// Mitsubishi GX Works2 project: miniproject_finalcode   PLC: Q03UDV

PROGRAM MAIN
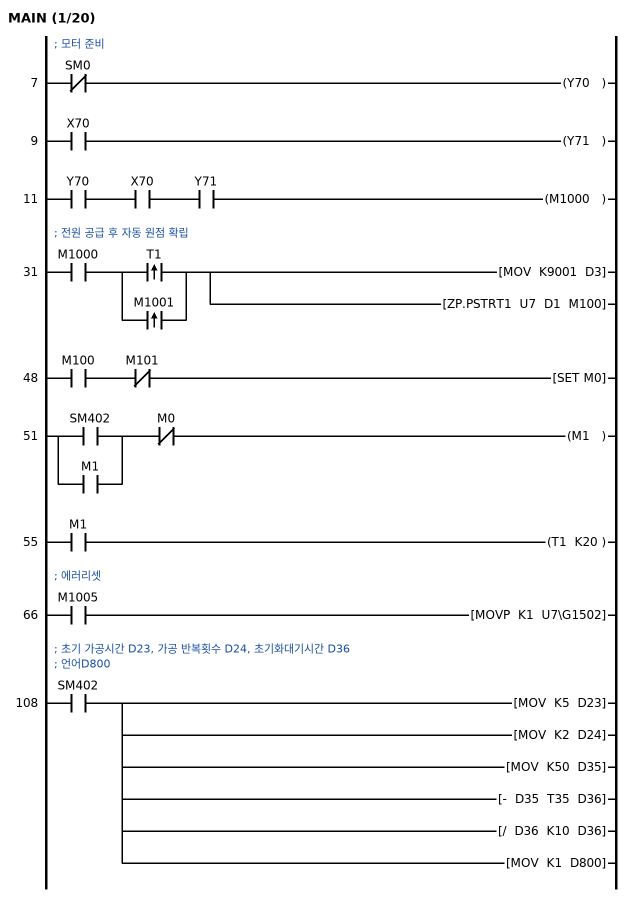
; 모터 준비
7     LDI     SM0
      OUT     Y70
9     LD      X70
      OUT     Y71
11    LD      Y70
      AND     X70
      AND     Y71
      OUT     M1000
; 전원 공급 후 자동 원점 확립
31    LD      M1000
      LDP     T1
      ORP     M1001
      ANB
      MOV     K9001 D3
      ZP.PSTRT1 U7 D1 M100
48    LD      M100
      ANI     M101
      SET     M0
51    LD      SM402
      OR      M1
      ANI     M0
      OUT     M1
55    LD      M1
      OUT     T1 K20
; 에러리셋
66    LD      M1005
      MOVP    K1 U7\G1502
; 초기 가공시간 D23, 가공 반복횟수 D24, 초기화대기시간 D36
; 언어D800
108   LD      SM402
      MOV     K5 D23
      MOV     K2 D24
      MOV     K50 D35
      -       D35 T35 D36
      /       D36 K10 D36
      MOV     K1 D800
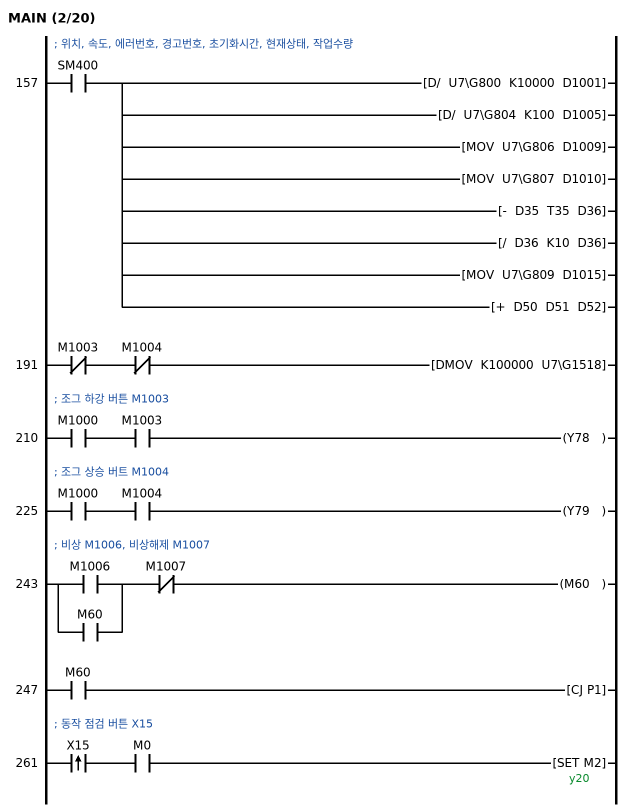
; 위치, 속도, 에러번호, 경고번호, 초기화시간, 현재상태, 작업수량
157   LD      SM400
      D/      U7\G800 K10000 D1001
      D/      U7\G804 K100 D1005
      MOV     U7\G806 D1009
      MOV     U7\G807 D1010
      -       D35 T35 D36
      /       D36 K10 D36
      MOV     U7\G809 D1015
      +       D50 D51 D52
191   LDI     M1003
      ANI     M1004
      DMOV    K100000 U7\G1518
; 조그 하강 버튼 M1003
210   LD      M1000
      AND     M1003
      OUT     Y78
; 조그 상승 버트 M1004
225   LD      M1000
      AND     M1004
      OUT     Y79
; 비상 M1006, 비상해제 M1007
243   LD      M1006
      OR      M60
      ANI     M1007
      OUT     M60
247   LD      M60
      CJ      P1
; 동작 점검 버튼 X15
261   LDP     X15
      AND     M0
      SET     M2  ; y20
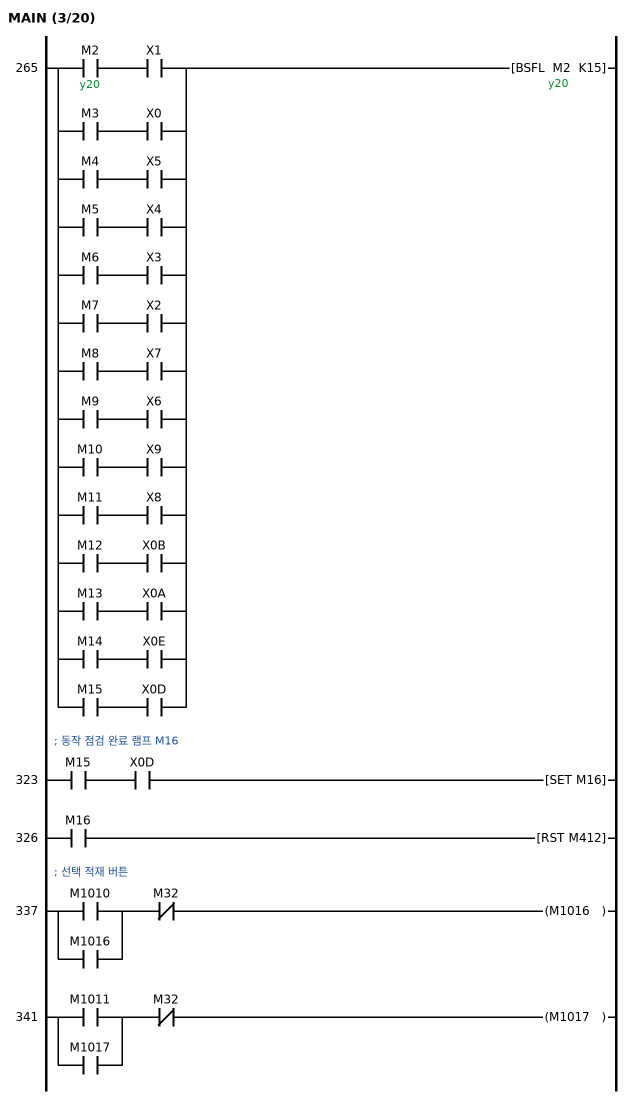
265   LD      M2  ; y20
      AND     X1
      LD      M3
      AND     X0
      ORB
      LD      M4
      AND     X5
      ORB
      LD      M5
      AND     X4
      ORB
      LD      M6
      AND     X3
      ORB
      LD      M7
      AND     X2
      ORB
      LD      M8
      AND     X7
      ORB
      LD      M9
      AND     X6
      ORB
      LD      M10
      AND     X9
      ORB
      LD      M11
      AND     X8
      ORB
      LD      M12
      AND     X0B
      ORB
      LD      M13
      AND     X0A
      ORB
      LD      M14
      AND     X0E
      ORB
      LD      M15
      AND     X0D
      ORB
      BSFL    M2 K15
; 동작 점검 완료 램프 M16
323   LD      M15
      AND     X0D
      SET     M16
326   LD      M16
      RST     M412
; 선택 적재 버튼
337   LD      M1010
      OR      M1016
      ANI     M32
      OUT     M1016
341   LD      M1011
      OR      M1017
      ANI     M32
      OUT     M1017
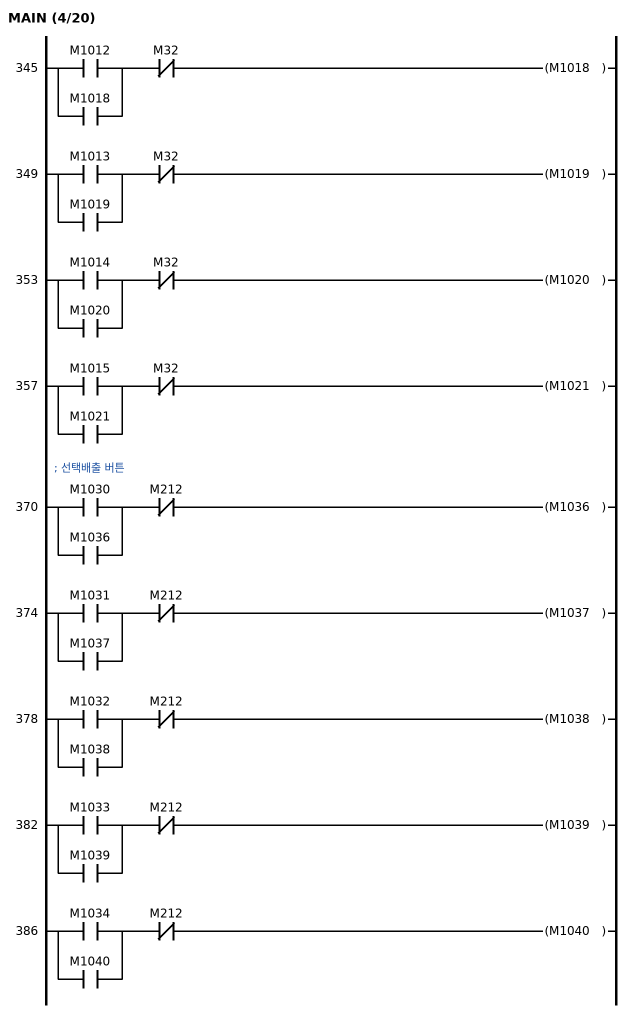
345   LD      M1012
      OR      M1018
      ANI     M32
      OUT     M1018
349   LD      M1013
      OR      M1019
      ANI     M32
      OUT     M1019
353   LD      M1014
      OR      M1020
      ANI     M32
      OUT     M1020
357   LD      M1015
      OR      M1021
      ANI     M32
      OUT     M1021
; 선택배출 버튼
370   LD      M1030
      OR      M1036
      ANI     M212
      OUT     M1036
374   LD      M1031
      OR      M1037
      ANI     M212
      OUT     M1037
378   LD      M1032
      OR      M1038
      ANI     M212
      OUT     M1038
382   LD      M1033
      OR      M1039
      ANI     M212
      OUT     M1039
386   LD      M1034
      OR      M1040
      ANI     M212
      OUT     M1040
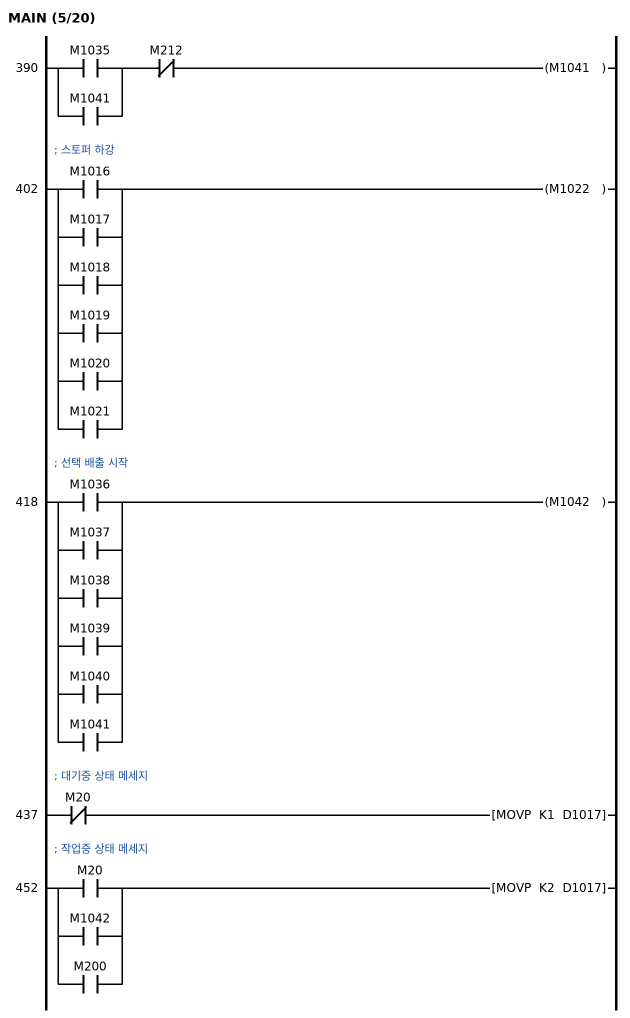
390   LD      M1035
      OR      M1041
      ANI     M212
      OUT     M1041
; 스토퍼 하강
402   LD      M1016
      OR      M1017
      OR      M1018
      OR      M1019
      OR      M1020
      OR      M1021
      OUT     M1022
; 선택 배출 시작
418   LD      M1036
      OR      M1037
      OR      M1038
      OR      M1039
      OR      M1040
      OR      M1041
      OUT     M1042
; 대기중 상태 메세지
437   LDI     M20
      MOVP    K1 D1017
; 작업중 상태 메세지
452   LD      M20
      OR      M1042
      OR      M200
      MOVP    K2 D1017
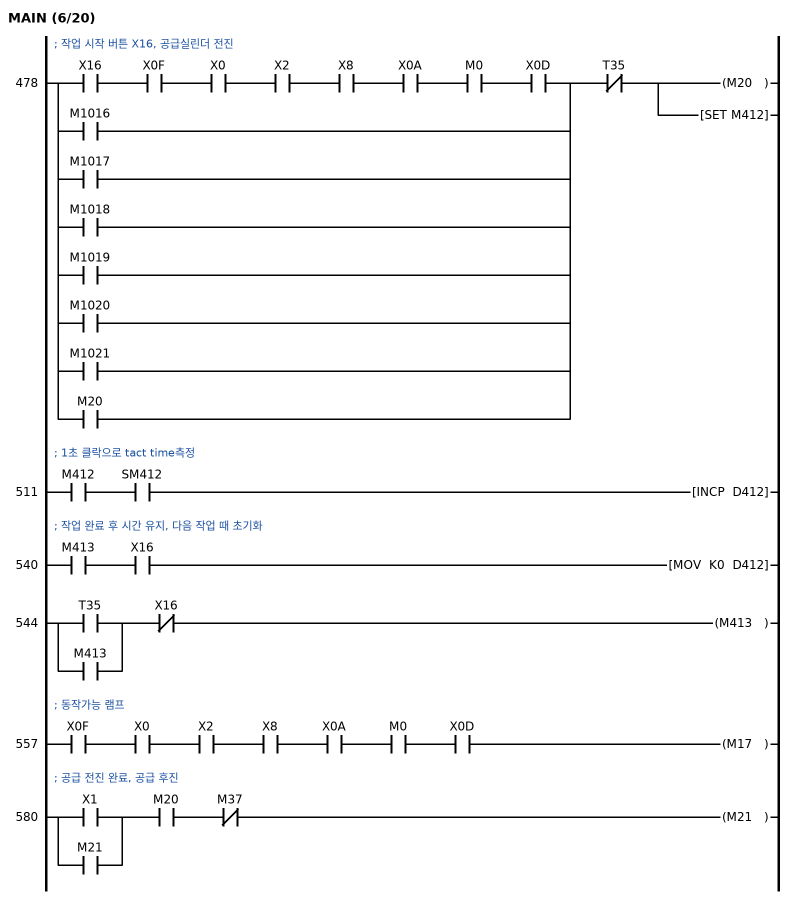
; 작업 시작 버튼 X16, 공급실린더 전진
478   LD      X16
      AND     X0F
      AND     X0
      AND     X2
      AND     X8
      AND     X0A
      AND     M0
      AND     X0D
      OR      M1016
      OR      M1017
      OR      M1018
      OR      M1019
      OR      M1020
      OR      M1021
      OR      M20
      ANI     T35
      OUT     M20
      SET     M412
; 1초 클락으로 tact time측정
511   LD      M412
      AND     SM412
      INCP    D412
; 작업 완료 후 시간 유지, 다음 작업 때 초기화
540   LD      M413
      AND     X16
      MOV     K0 D412
544   LD      T35
      OR      M413
      ANI     X16
      OUT     M413
; 동작가능 램프
557   LD      X0F
      AND     X0
      AND     X2
      AND     X8
      AND     X0A
      AND     M0
      AND     X0D
      OUT     M17
; 공급 전진 완료, 공급 후진
580   LD      X1
      OR      M21
      AND     M20
      ANI     M37
      OUT     M21
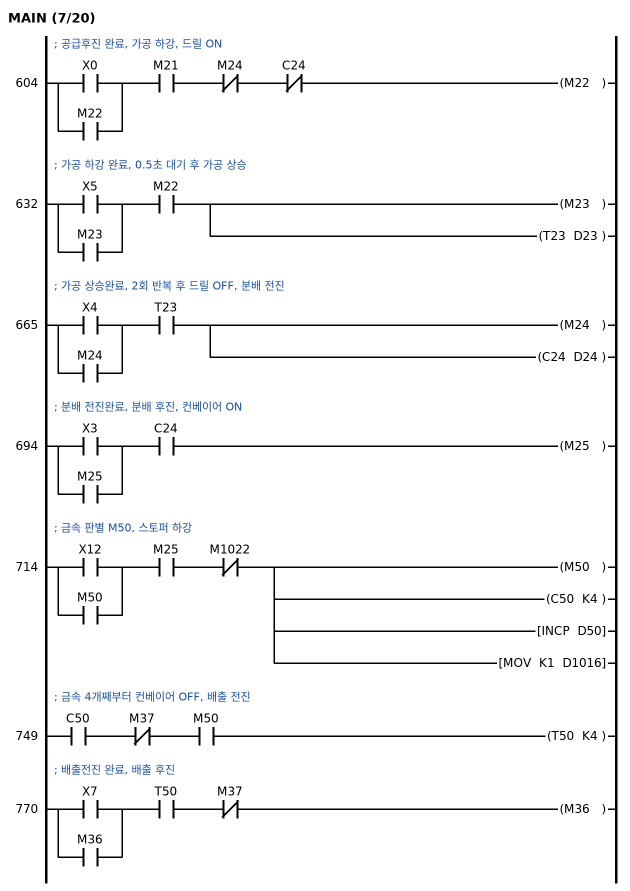
; 공급후진 완료, 가공 하강, 드릴 ON
604   LD      X0
      OR      M22
      AND     M21
      ANI     M24
      ANI     C24
      OUT     M22
; 가공 하강 완료, 0.5초 대기 후 가공 상승
632   LD      X5
      OR      M23
      AND     M22
      OUT     M23
      OUT     T23 D23
; 가공 상승완료, 2회 반복 후 드릴 OFF, 분배 전진
665   LD      X4
      OR      M24
      AND     T23
      OUT     M24
      OUT     C24 D24
; 분배 전진완료, 분배 후진, 컨베이어 ON
694   LD      X3
      OR      M25
      AND     C24
      OUT     M25
; 금속 판별 M50, 스토퍼 하강
714   LD      X12
      OR      M50
      AND     M25
      ANI     M1022
      OUT     M50
      OUT     C50 K4
      INCP    D50
      MOV     K1 D1016
; 금속 4개째부터 컨베이어 OFF, 배출 전진
749   LD      C50
      ANI     M37
      AND     M50
      OUT     T50 K4
; 배출전진 완료, 배출 후진
770   LD      X7
      OR      M36
      AND     T50
      ANI     M37
      OUT     M36
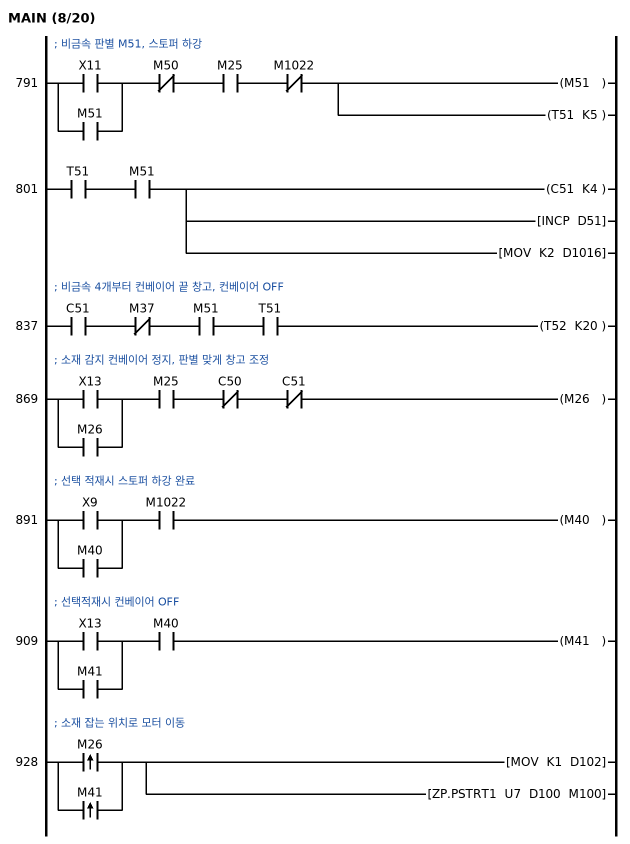
; 비금속 판별 M51, 스토퍼 하강
791   LD      X11
      OR      M51
      ANI     M50
      AND     M25
      ANI     M1022
      OUT     M51
      OUT     T51 K5
801   LD      T51
      AND     M51
      OUT     C51 K4
      INCP    D51
      MOV     K2 D1016
; 비금속 4개부터 컨베이어 끝 창고, 컨베이어 OFF
837   LD      C51
      ANI     M37
      AND     M51
      AND     T51
      OUT     T52 K20
; 소재 감지 컨베이어 정지, 판별 맞게 창고 조정
869   LD      X13
      OR      M26
      AND     M25
      ANI     C50
      ANI     C51
      OUT     M26
; 선택 적재시 스토퍼 하강 완료
891   LD      X9
      OR      M40
      AND     M1022
      OUT     M40
; 선택적재시 컨베이어 OFF
909   LD      X13
      OR      M41
      AND     M40
      OUT     M41
; 소재 잡는 위치로 모터 이동
928   LDP     M26
      ORP     M41
      MOV     K1 D102
      ZP.PSTRT1 U7 D100 M100
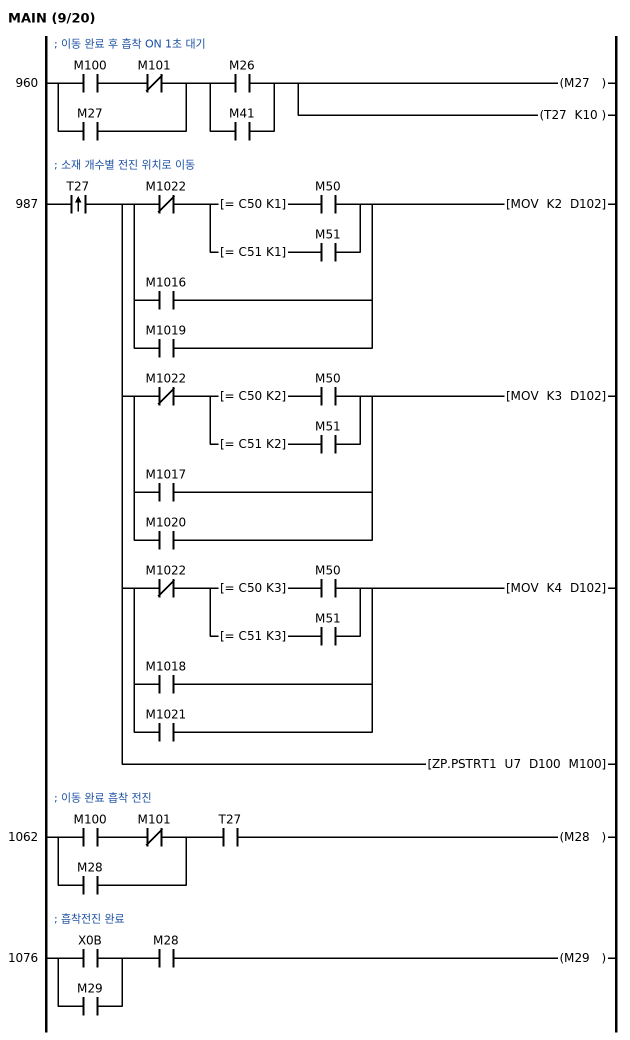
; 이동 완료 후 흡착 ON 1초 대기
960   LD      M100
      ANI     M101
      OR      M27
      LD      M26
      OR      M41
      ANB
      OUT     M27
      OUT     T27 K10
; 소재 개수별 전진 위치로 이동
987   LDP     T27
      MPS
      LDI     M1022
      LD=     C50 K1
      AND     M50
      LD=     C51 K1
      AND     M51
      ORB
      ANB
      OR      M1016
      OR      M1019
      ANB
      MOV     K2 D102
      MRD
      LDI     M1022
      LD=     C50 K2
      AND     M50
      LD=     C51 K2
      AND     M51
      ORB
      ANB
      OR      M1017
      OR      M1020
      ANB
      MOV     K3 D102
      MRD
      LDI     M1022
      LD=     C50 K3
      AND     M50
      LD=     C51 K3
      AND     M51
      ORB
      ANB
      OR      M1018
      OR      M1021
      ANB
      MOV     K4 D102
      MPP
      ZP.PSTRT1 U7 D100 M100
; 이동 완료 흡착 전진
1062  LD      M100
      ANI     M101
      OR      M28
      AND     T27
      OUT     M28
; 흡착전진 완료
1076  LD      X0B
      OR      M29
      AND     M28
      OUT     M29
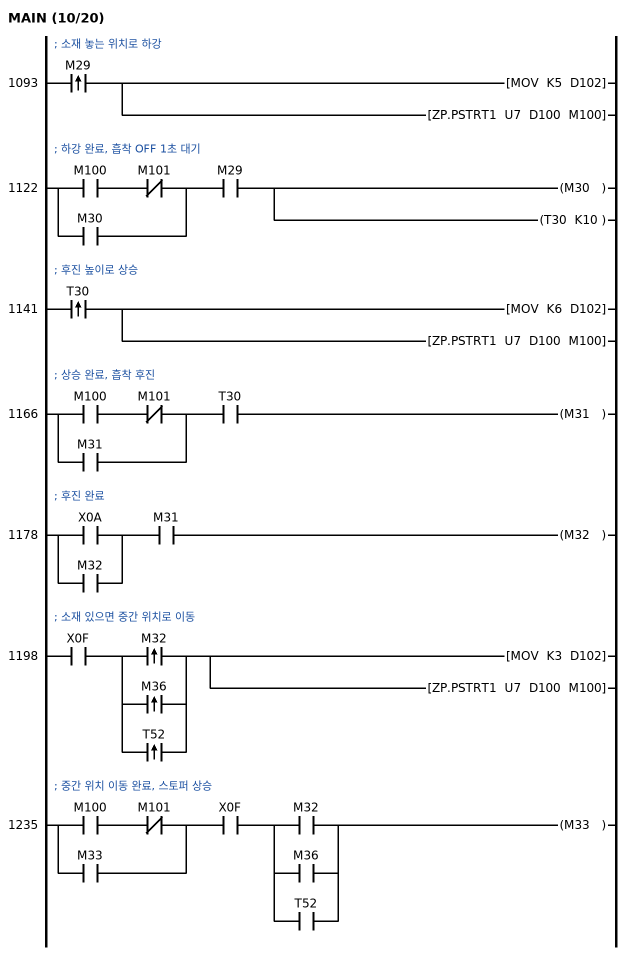
; 소재 놓는 위치로 하강
1093  LDP     M29
      MOV     K5 D102
      ZP.PSTRT1 U7 D100 M100
; 하강 완료, 흡착 OFF 1초 대기
1122  LD      M100
      ANI     M101
      OR      M30
      AND     M29
      OUT     M30
      OUT     T30 K10
; 후진 높이로 상승
1141  LDP     T30
      MOV     K6 D102
      ZP.PSTRT1 U7 D100 M100
; 상승 완료, 흡착 후진
1166  LD      M100
      ANI     M101
      OR      M31
      AND     T30
      OUT     M31
; 후진 완료
1178  LD      X0A
      OR      M32
      AND     M31
      OUT     M32
; 소재 있으면 중간 위치로 이동
1198  LD      X0F
      LDP     M32
      ORP     M36
      ORP     T52
      ANB
      MOV     K3 D102
      ZP.PSTRT1 U7 D100 M100
; 중간 위치 이동 완료, 스토퍼 상승
1235  LD      M100
      ANI     M101
      OR      M33
      AND     X0F
      LD      M32
      OR      M36
      OR      T52
      ANB
      OUT     M33
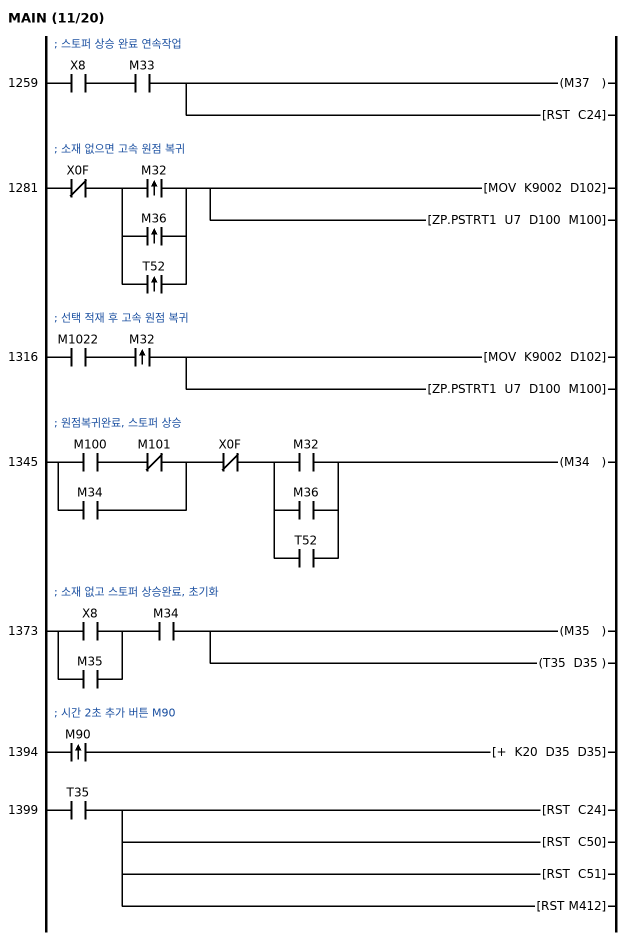
; 스토퍼 상승 완료 연속작업
1259  LD      X8
      AND     M33
      OUT     M37
      RST     C24
; 소재 없으면 고속 원점 복귀
1281  LDI     X0F
      LDP     M32
      ORP     M36
      ORP     T52
      ANB
      MOV     K9002 D102
      ZP.PSTRT1 U7 D100 M100
; 선택 적재 후 고속 원점 복귀
1316  LD      M1022
      ANDP    M32
      MOV     K9002 D102
      ZP.PSTRT1 U7 D100 M100
; 원점복귀완료, 스토퍼 상승
1345  LD      M100
      ANI     M101
      OR      M34
      ANI     X0F
      LD      M32
      OR      M36
      OR      T52
      ANB
      OUT     M34
; 소재 없고 스토퍼 상승완료, 초기화
1373  LD      X8
      OR      M35
      AND     M34
      OUT     M35
      OUT     T35 D35
; 시간 2초 추가 버튼 M90
1394  LDP     M90
      +       K20 D35 D35
1399  LD      T35
      RST     C24
      RST     C50
      RST     C51
      RST     M412
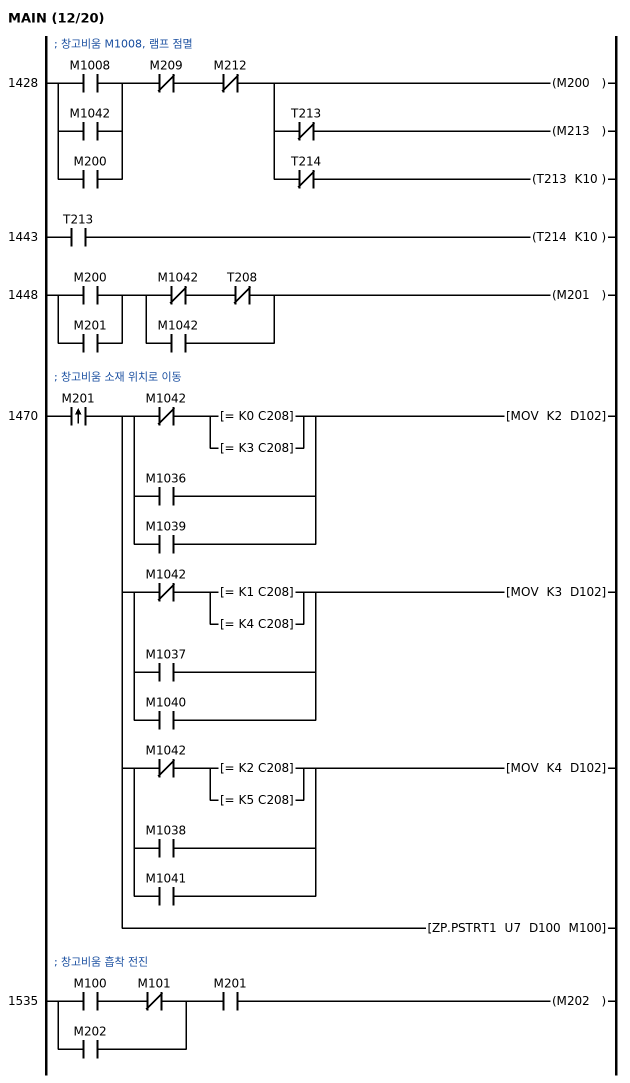
; 창고비움 M1008, 램프 점멸
1428  LD      M1008
      OR      M1042
      OR      M200
      ANI     M209
      ANI     M212
      OUT     M200
      MPS
      ANI     T213
      OUT     M213
      MPP
      ANI     T214
      OUT     T213 K10
1443  LD      T213
      OUT     T214 K10
1448  LD      M200
      OR      M201
      LDI     M1042
      ANI     T208
      OR      M1042
      ANB
      OUT     M201
; 창고비움 소재 위치로 이동
1470  LDP     M201
      MPS
      LDI     M1042
      LD=     K0 C208
      OR=     K3 C208
      ANB
      OR      M1036
      OR      M1039
      ANB
      MOV     K2 D102
      MRD
      LDI     M1042
      LD=     K1 C208
      OR=     K4 C208
      ANB
      OR      M1037
      OR      M1040
      ANB
      MOV     K3 D102
      MRD
      LDI     M1042
      LD=     K2 C208
      OR=     K5 C208
      ANB
      OR      M1038
      OR      M1041
      ANB
      MOV     K4 D102
      MPP
      ZP.PSTRT1 U7 D100 M100
; 창고비움 흡착 전진
1535  LD      M100
      ANI     M101
      OR      M202
      AND     M201
      OUT     M202
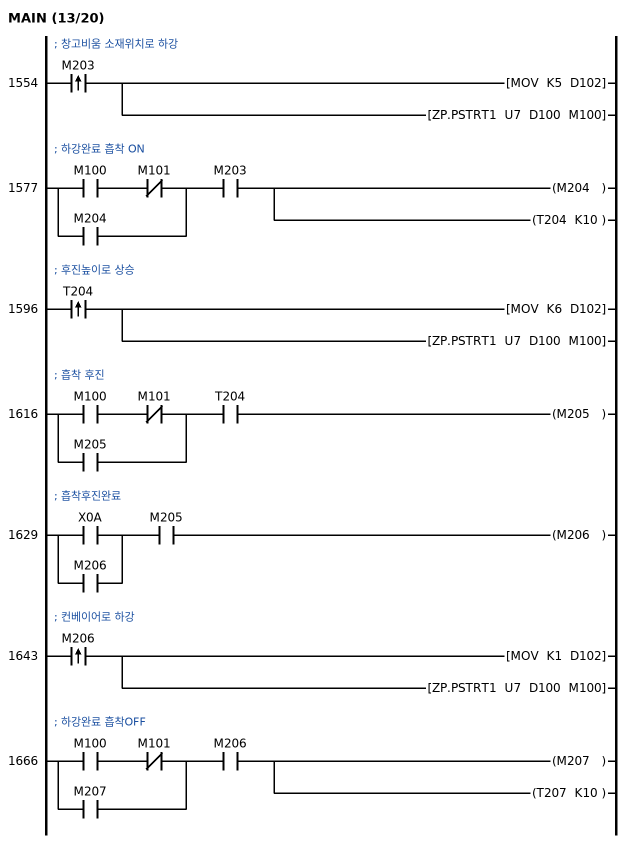
; 창고비움 소재위치로 하강
1554  LDP     M203
      MOV     K5 D102
      ZP.PSTRT1 U7 D100 M100
; 하강완료 흡착 ON
1577  LD      M100
      ANI     M101
      OR      M204
      AND     M203
      OUT     M204
      OUT     T204 K10
; 후진높이로 상승
1596  LDP     T204
      MOV     K6 D102
      ZP.PSTRT1 U7 D100 M100
; 흡착 후진
1616  LD      M100
      ANI     M101
      OR      M205
      AND     T204
      OUT     M205
; 흡착후진완료
1629  LD      X0A
      OR      M206
      AND     M205
      OUT     M206
; 컨베이어로 하강
1643  LDP     M206
      MOV     K1 D102
      ZP.PSTRT1 U7 D100 M100
; 하강완료 흡착OFF
1666  LD      M100
      ANI     M101
      OR      M207
      AND     M206
      OUT     M207
      OUT     T207 K10
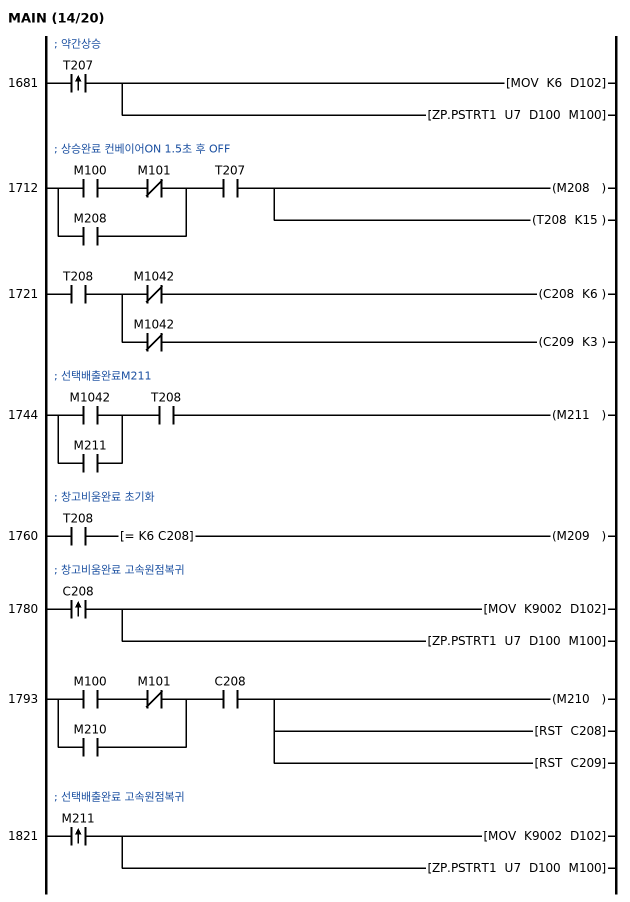
; 약간상승
1681  LDP     T207
      MOV     K6 D102
      ZP.PSTRT1 U7 D100 M100
; 상승완료 컨베이어ON 1.5초 후 OFF
1712  LD      M100
      ANI     M101
      OR      M208
      AND     T207
      OUT     M208
      OUT     T208 K15
1721  LD      T208
      MPS
      ANI     M1042
      OUT     C208 K6
      MPP
      ANI     M1042
      OUT     C209 K3
; 선택배출완료M211
1744  LD      M1042
      OR      M211
      AND     T208
      OUT     M211
; 창고비움완료 초기화
1760  LD      T208
      AND=    K6 C208
      OUT     M209
; 창고비움완료 고속원점복귀
1780  LDP     C208
      MOV     K9002 D102
      ZP.PSTRT1 U7 D100 M100
1793  LD      M100
      ANI     M101
      OR      M210
      AND     C208
      OUT     M210
      RST     C208
      RST     C209
; 선택배출완료 고속원점복귀
1821  LDP     M211
      MOV     K9002 D102
      ZP.PSTRT1 U7 D100 M100
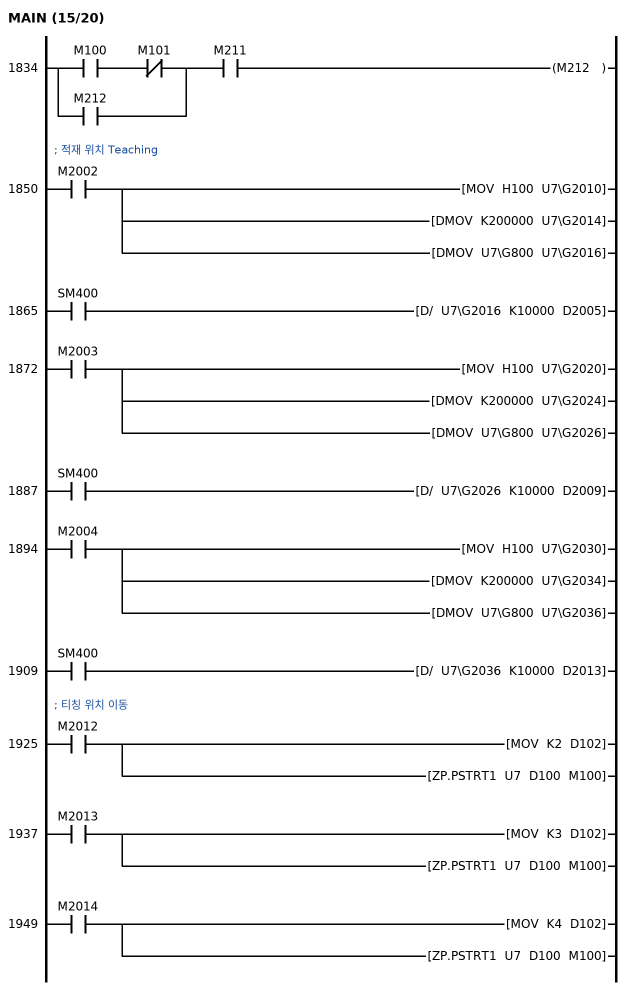
1834  LD      M100
      ANI     M101
      OR      M212
      AND     M211
      OUT     M212
; 적재 위치 Teaching
1850  LD      M2002
      MOV     H100 U7\G2010
      DMOV    K200000 U7\G2014
      DMOV    U7\G800 U7\G2016
1865  LD      SM400
      D/      U7\G2016 K10000 D2005
1872  LD      M2003
      MOV     H100 U7\G2020
      DMOV    K200000 U7\G2024
      DMOV    U7\G800 U7\G2026
1887  LD      SM400
      D/      U7\G2026 K10000 D2009
1894  LD      M2004
      MOV     H100 U7\G2030
      DMOV    K200000 U7\G2034
      DMOV    U7\G800 U7\G2036
1909  LD      SM400
      D/      U7\G2036 K10000 D2013
; 티칭 위치 이동
1925  LD      M2012
      MOV     K2 D102
      ZP.PSTRT1 U7 D100 M100
1937  LD      M2013
      MOV     K3 D102
      ZP.PSTRT1 U7 D100 M100
1949  LD      M2014
      MOV     K4 D102
      ZP.PSTRT1 U7 D100 M100
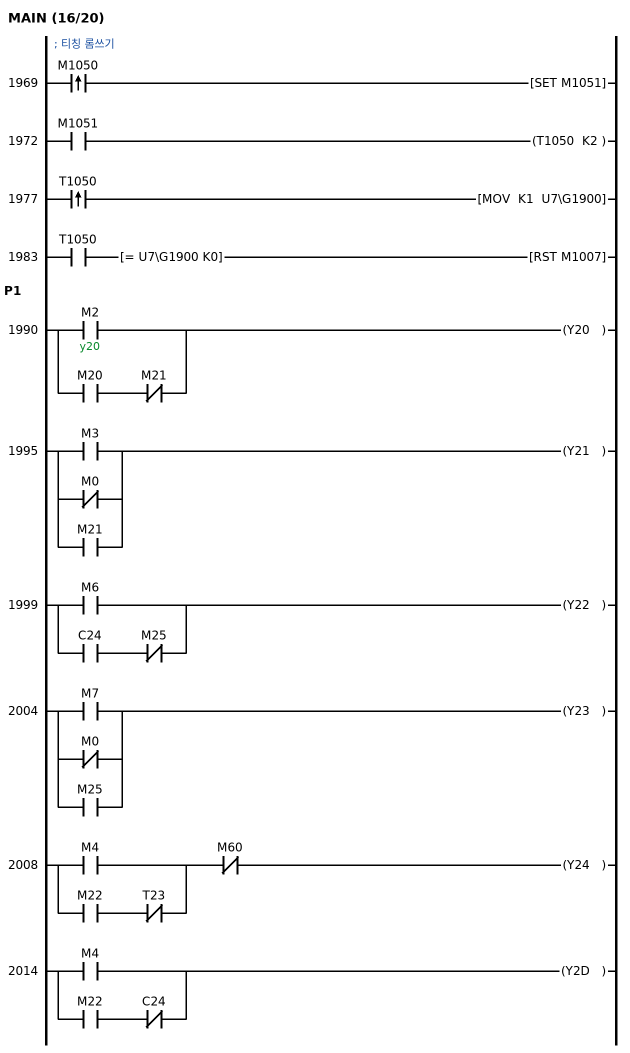
; 티칭 롬쓰기
1969  LDP     M1050
      SET     M1051
1972  LD      M1051
      OUT     T1050 K2
1977  LDP     T1050
      MOV     K1 U7\G1900
1983  LD      T1050
      AND=    U7\G1900 K0
      RST     M1007
      P1
1990  LD      M2  ; y20
      LD      M20
      ANI     M21
      ORB
      OUT     Y20
1995  LD      M3
      ORI     M0
      OR      M21
      OUT     Y21
1999  LD      M6
      LD      C24
      ANI     M25
      ORB
      OUT     Y22
2004  LD      M7
      ORI     M0
      OR      M25
      OUT     Y23
2008  LD      M4
      LD      M22
      ANI     T23
      ORB
      ANI     M60
      OUT     Y24
2014  LD      M4
      LD      M22
      ANI     C24
      ORB
      OUT     Y2D
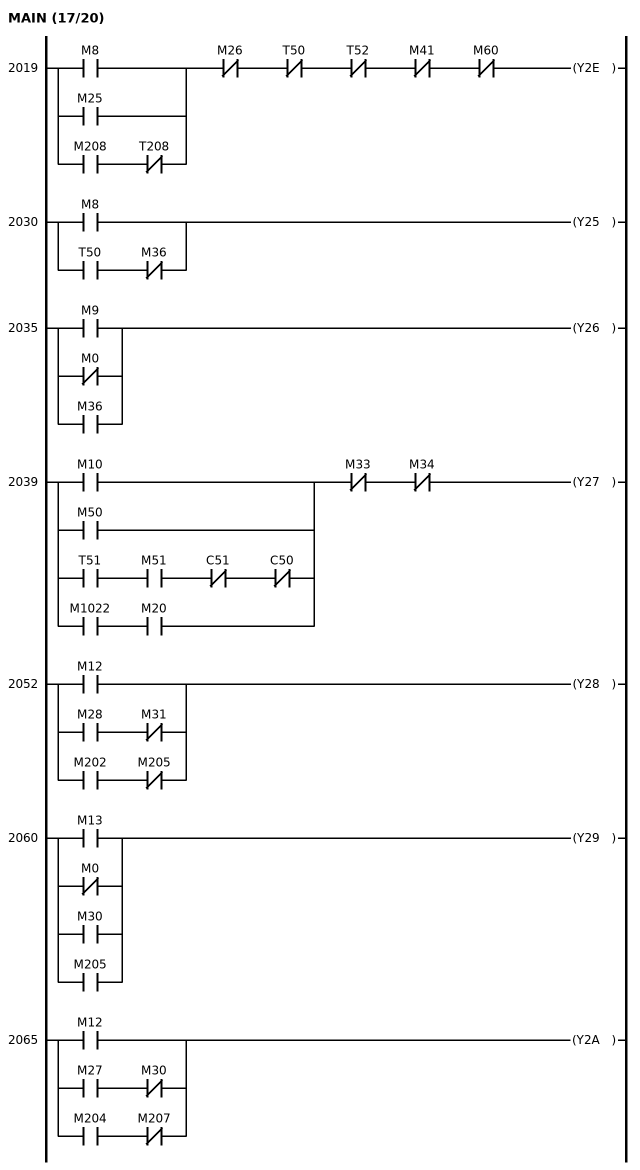
2019  LD      M8
      OR      M25
      LD      M208
      ANI     T208
      ORB
      ANI     M26
      ANI     T50
      ANI     T52
      ANI     M41
      ANI     M60
      OUT     Y2E
2030  LD      M8
      LD      T50
      ANI     M36
      ORB
      OUT     Y25
2035  LD      M9
      ORI     M0
      OR      M36
      OUT     Y26
2039  LD      M10
      OR      M50
      LD      T51
      AND     M51
      ANI     C51
      ANI     C50
      ORB
      LD      M1022
      AND     M20
      ORB
      ANI     M33
      ANI     M34
      OUT     Y27
2052  LD      M12
      LD      M28
      ANI     M31
      ORB
      LD      M202
      ANI     M205
      ORB
      OUT     Y28
2060  LD      M13
      ORI     M0
      OR      M30
      OR      M205
      OUT     Y29
2065  LD      M12
      LD      M27
      ANI     M30
      ORB
      LD      M204
      ANI     M207
      ORB
      OUT     Y2A
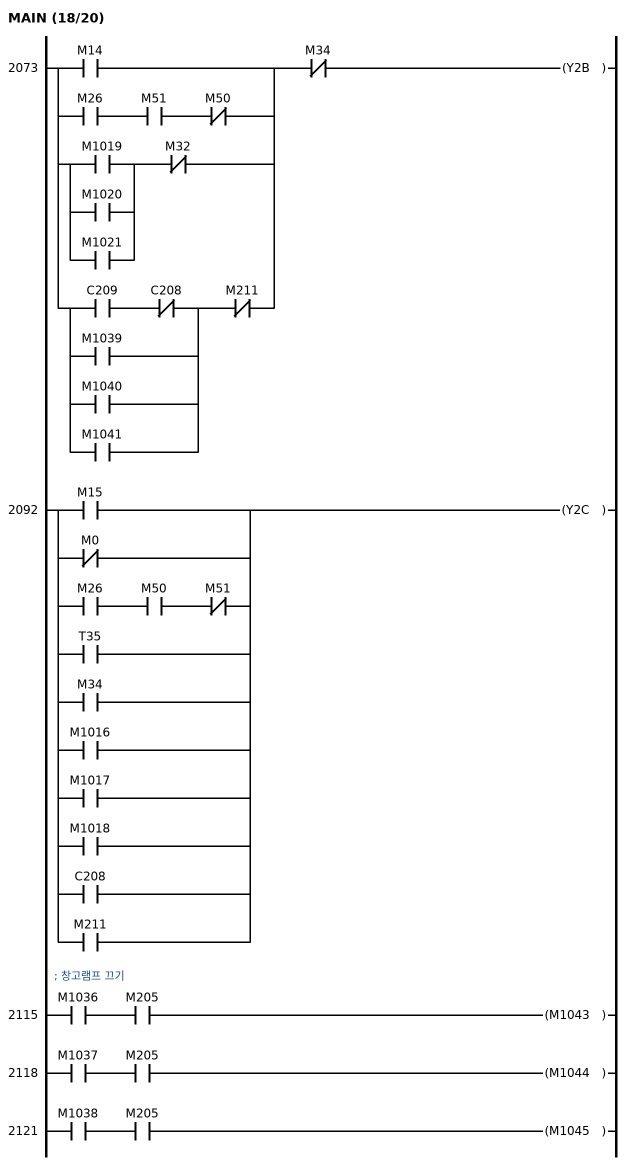
2073  LD      M14
      LD      M26
      AND     M51
      ANI     M50
      ORB
      LD      M1019
      OR      M1020
      OR      M1021
      ANI     M32
      ORB
      LD      C209
      ANI     C208
      OR      M1039
      OR      M1040
      OR      M1041
      ANI     M211
      ORB
      ANI     M34
      OUT     Y2B
2092  LD      M15
      ORI     M0
      LD      M26
      AND     M50
      ANI     M51
      ORB
      OR      T35
      OR      M34
      OR      M1016
      OR      M1017
      OR      M1018
      OR      C208
      OR      M211
      OUT     Y2C
; 창고램프 끄기
2115  LD      M1036
      AND     M205
      OUT     M1043
2118  LD      M1037
      AND     M205
      OUT     M1044
2121  LD      M1038
      AND     M205
      OUT     M1045
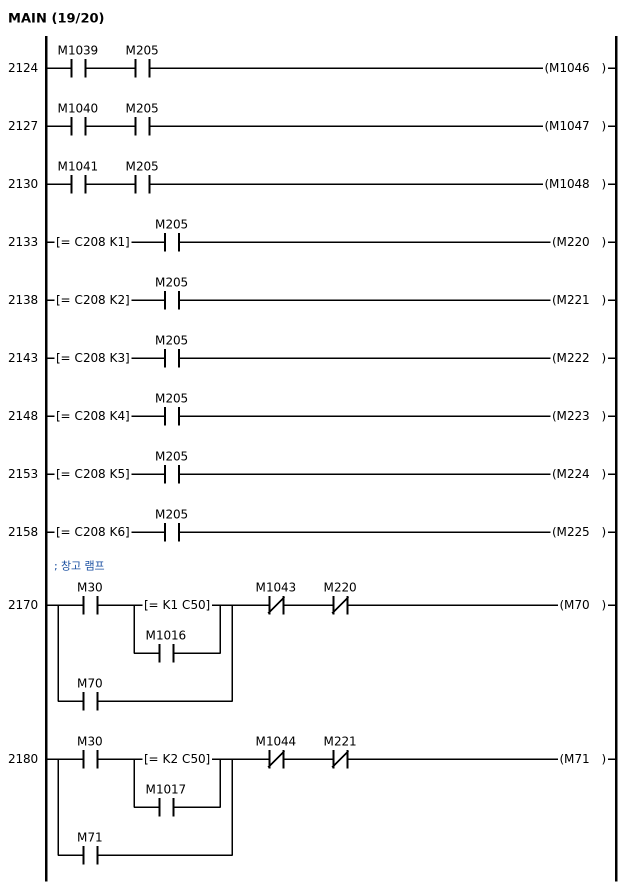
2124  LD      M1039
      AND     M205
      OUT     M1046
2127  LD      M1040
      AND     M205
      OUT     M1047
2130  LD      M1041
      AND     M205
      OUT     M1048
2133  LD=     C208 K1
      AND     M205
      OUT     M220
2138  LD=     C208 K2
      AND     M205
      OUT     M221
2143  LD=     C208 K3
      AND     M205
      OUT     M222
2148  LD=     C208 K4
      AND     M205
      OUT     M223
2153  LD=     C208 K5
      AND     M205
      OUT     M224
2158  LD=     C208 K6
      AND     M205
      OUT     M225
; 창고 램프
2170  LD      M30
      LD=     K1 C50
      OR      M1016
      ANB
      OR      M70
      ANI     M1043
      ANI     M220
      OUT     M70
2180  LD      M30
      LD=     K2 C50
      OR      M1017
      ANB
      OR      M71
      ANI     M1044
      ANI     M221
      OUT     M71
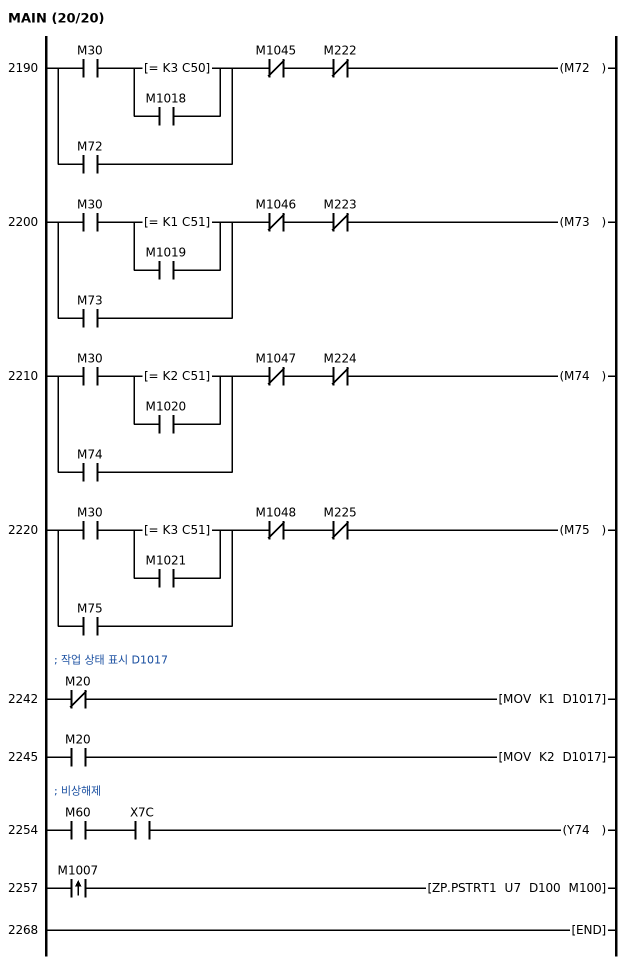
2190  LD      M30
      LD=     K3 C50
      OR      M1018
      ANB
      OR      M72
      ANI     M1045
      ANI     M222
      OUT     M72
2200  LD      M30
      LD=     K1 C51
      OR      M1019
      ANB
      OR      M73
      ANI     M1046
      ANI     M223
      OUT     M73
2210  LD      M30
      LD=     K2 C51
      OR      M1020
      ANB
      OR      M74
      ANI     M1047
      ANI     M224
      OUT     M74
2220  LD      M30
      LD=     K3 C51
      OR      M1021
      ANB
      OR      M75
      ANI     M1048
      ANI     M225
      OUT     M75
; 작업 상태 표시 D1017
2242  LDI     M20
      MOV     K1 D1017
2245  LD      M20
      MOV     K2 D1017
; 비상해제
2254  LD      M60
      AND     X7C
      OUT     Y74
2257  LDP     M1007
      ZP.PSTRT1 U7 D100 M100
2268  END
END_PROGRAM
